(* IEC 61131-3 sources: AXOpen/src/components.mitsubishi.robotics/app/src/IO/PLC_LINE, 7 files *)

(* ---- HwIdentifiers.st ---- *)
TYPE
    HwIdentifiers : WORD
    (
        PROFINET_IO_System_HwID :=	WORD#256,
        TZ535_PN_HwID :=	WORD#260,
        TZ535_PN_In_Out_64_byte_1_In_Out__64_byte_HwID :=	WORD#263,
        TZ535_PN_Rack_HwID :=	WORD#261,
        TZ535_PN_TZ535_PN_HwID :=	WORD#262,
        TZ535_PN_TZ535_PN_2D_TZ535_PNPROFINET_IO_HwID :=	WORD#264,
        TZ535_PN_TZ535_PN_profinet_HwID :=	WORD#257,
        TZ535_PN_TZ535_PN_profinet_Port_1_HwID :=	WORD#258,
        TZ535_PN_TZ535_PN_profinet_Port_2_HwID :=	WORD#259,
        plc_line_HwID :=	WORD#32,
        plc_line_Rail_0_HwID :=	WORD#265,
        plc_line_plc_line_HwID :=	WORD#48,
        plc_line_plc_line__plc_line_HwID :=	WORD#49,
        plc_line_plc_line_CPU_display_1_HwID :=	WORD#54,
        plc_line_plc_line_CPU_exec_unit_1_HwID :=	WORD#52,
        plc_line_plc_line_Card_reader_writer_1_HwID :=	WORD#51,
        plc_line_plc_line_DP_interface_1_HwID :=	WORD#60,
        plc_line_plc_line_LicenseManager_1_HwID :=	WORD#42,
        plc_line_plc_line_OPC_UA_1_HwID :=	WORD#117,
        plc_line_plc_line_PROFINET_interface_2_HwID :=	WORD#72,
        plc_line_plc_line_PROFINET_interface_2_Port_1_HwID :=	WORD#73,
        plc_line_plc_line_Virtual_communication_interface_HwID :=	WORD#135,
        plc_line_plc_line_plc_line_HwID :=	WORD#50,
        plc_line_plc_line_profinet_x1_HwID :=	WORD#64,
        plc_line_plc_line_profinet_x1_Port1_HwID :=	WORD#65,
        plc_line_plc_line_profinet_x1_Port2_HwID :=	WORD#66,

        NONE := WORD#0
    );
END_TYPE

(* ---- HwInputs.st ---- *)
TYPE
	HwInputs : STRUCT
		TZ535_PN_In_Out_64_byte_1 AT %B0 : ARRAY[0..63] OF BYTE;
	END_STRUCT;
END_TYPE

(* ---- HwOutputs.st ---- *)
TYPE
	HwOutputs : STRUCT
		TZ535_PN_In_Out_64_byte_1 AT %B0 : ARRAY[0..63] OF BYTE;
	END_STRUCT;
END_TYPE

(* ---- PlcInputs.st ---- *)
TYPE
	PlcInputs : STRUCT
		TZ535_PN_In_Out_64_byte_1 : ARRAY[0..63] OF BYTE;
	END_STRUCT;
END_TYPE

(* ---- PlcOutputs.st ---- *)
TYPE
	PlcOutputs : STRUCT
		TZ535_PN_In_Out_64_byte_1 : ARRAY[0..63] OF BYTE;
	END_STRUCT;
END_TYPE

(* ---- CopyInputs.st ---- *)
FUNCTION CopyInputs
	VAR_EXTERNAL
		HwInputs : HwInputs;
		PlcInputs : PlcInputs;
	END_VAR
	PlcInputs.TZ535_PN_In_Out_64_byte_1[0] := HwInputs.TZ535_PN_In_Out_64_byte_1[0];
	PlcInputs.TZ535_PN_In_Out_64_byte_1[1] := HwInputs.TZ535_PN_In_Out_64_byte_1[1];
	PlcInputs.TZ535_PN_In_Out_64_byte_1[2] := HwInputs.TZ535_PN_In_Out_64_byte_1[2];
	PlcInputs.TZ535_PN_In_Out_64_byte_1[3] := HwInputs.TZ535_PN_In_Out_64_byte_1[3];
	PlcInputs.TZ535_PN_In_Out_64_byte_1[4] := HwInputs.TZ535_PN_In_Out_64_byte_1[4];
	PlcInputs.TZ535_PN_In_Out_64_byte_1[5] := HwInputs.TZ535_PN_In_Out_64_byte_1[5];
	PlcInputs.TZ535_PN_In_Out_64_byte_1[6] := HwInputs.TZ535_PN_In_Out_64_byte_1[6];
	PlcInputs.TZ535_PN_In_Out_64_byte_1[7] := HwInputs.TZ535_PN_In_Out_64_byte_1[7];
	PlcInputs.TZ535_PN_In_Out_64_byte_1[8] := HwInputs.TZ535_PN_In_Out_64_byte_1[8];
	PlcInputs.TZ535_PN_In_Out_64_byte_1[9] := HwInputs.TZ535_PN_In_Out_64_byte_1[9];
	PlcInputs.TZ535_PN_In_Out_64_byte_1[10] := HwInputs.TZ535_PN_In_Out_64_byte_1[10];
	PlcInputs.TZ535_PN_In_Out_64_byte_1[11] := HwInputs.TZ535_PN_In_Out_64_byte_1[11];
	PlcInputs.TZ535_PN_In_Out_64_byte_1[12] := HwInputs.TZ535_PN_In_Out_64_byte_1[12];
	PlcInputs.TZ535_PN_In_Out_64_byte_1[13] := HwInputs.TZ535_PN_In_Out_64_byte_1[13];
	PlcInputs.TZ535_PN_In_Out_64_byte_1[14] := HwInputs.TZ535_PN_In_Out_64_byte_1[14];
	PlcInputs.TZ535_PN_In_Out_64_byte_1[15] := HwInputs.TZ535_PN_In_Out_64_byte_1[15];
	PlcInputs.TZ535_PN_In_Out_64_byte_1[16] := HwInputs.TZ535_PN_In_Out_64_byte_1[16];
	PlcInputs.TZ535_PN_In_Out_64_byte_1[17] := HwInputs.TZ535_PN_In_Out_64_byte_1[17];
	PlcInputs.TZ535_PN_In_Out_64_byte_1[18] := HwInputs.TZ535_PN_In_Out_64_byte_1[18];
	PlcInputs.TZ535_PN_In_Out_64_byte_1[19] := HwInputs.TZ535_PN_In_Out_64_byte_1[19];
	PlcInputs.TZ535_PN_In_Out_64_byte_1[20] := HwInputs.TZ535_PN_In_Out_64_byte_1[20];
	PlcInputs.TZ535_PN_In_Out_64_byte_1[21] := HwInputs.TZ535_PN_In_Out_64_byte_1[21];
	PlcInputs.TZ535_PN_In_Out_64_byte_1[22] := HwInputs.TZ535_PN_In_Out_64_byte_1[22];
	PlcInputs.TZ535_PN_In_Out_64_byte_1[23] := HwInputs.TZ535_PN_In_Out_64_byte_1[23];
	PlcInputs.TZ535_PN_In_Out_64_byte_1[24] := HwInputs.TZ535_PN_In_Out_64_byte_1[24];
	PlcInputs.TZ535_PN_In_Out_64_byte_1[25] := HwInputs.TZ535_PN_In_Out_64_byte_1[25];
	PlcInputs.TZ535_PN_In_Out_64_byte_1[26] := HwInputs.TZ535_PN_In_Out_64_byte_1[26];
	PlcInputs.TZ535_PN_In_Out_64_byte_1[27] := HwInputs.TZ535_PN_In_Out_64_byte_1[27];
	PlcInputs.TZ535_PN_In_Out_64_byte_1[28] := HwInputs.TZ535_PN_In_Out_64_byte_1[28];
	PlcInputs.TZ535_PN_In_Out_64_byte_1[29] := HwInputs.TZ535_PN_In_Out_64_byte_1[29];
	PlcInputs.TZ535_PN_In_Out_64_byte_1[30] := HwInputs.TZ535_PN_In_Out_64_byte_1[30];
	PlcInputs.TZ535_PN_In_Out_64_byte_1[31] := HwInputs.TZ535_PN_In_Out_64_byte_1[31];
	PlcInputs.TZ535_PN_In_Out_64_byte_1[32] := HwInputs.TZ535_PN_In_Out_64_byte_1[32];
	PlcInputs.TZ535_PN_In_Out_64_byte_1[33] := HwInputs.TZ535_PN_In_Out_64_byte_1[33];
	PlcInputs.TZ535_PN_In_Out_64_byte_1[34] := HwInputs.TZ535_PN_In_Out_64_byte_1[34];
	PlcInputs.TZ535_PN_In_Out_64_byte_1[35] := HwInputs.TZ535_PN_In_Out_64_byte_1[35];
	PlcInputs.TZ535_PN_In_Out_64_byte_1[36] := HwInputs.TZ535_PN_In_Out_64_byte_1[36];
	PlcInputs.TZ535_PN_In_Out_64_byte_1[37] := HwInputs.TZ535_PN_In_Out_64_byte_1[37];
	PlcInputs.TZ535_PN_In_Out_64_byte_1[38] := HwInputs.TZ535_PN_In_Out_64_byte_1[38];
	PlcInputs.TZ535_PN_In_Out_64_byte_1[39] := HwInputs.TZ535_PN_In_Out_64_byte_1[39];
	PlcInputs.TZ535_PN_In_Out_64_byte_1[40] := HwInputs.TZ535_PN_In_Out_64_byte_1[40];
	PlcInputs.TZ535_PN_In_Out_64_byte_1[41] := HwInputs.TZ535_PN_In_Out_64_byte_1[41];
	PlcInputs.TZ535_PN_In_Out_64_byte_1[42] := HwInputs.TZ535_PN_In_Out_64_byte_1[42];
	PlcInputs.TZ535_PN_In_Out_64_byte_1[43] := HwInputs.TZ535_PN_In_Out_64_byte_1[43];
	PlcInputs.TZ535_PN_In_Out_64_byte_1[44] := HwInputs.TZ535_PN_In_Out_64_byte_1[44];
	PlcInputs.TZ535_PN_In_Out_64_byte_1[45] := HwInputs.TZ535_PN_In_Out_64_byte_1[45];
	PlcInputs.TZ535_PN_In_Out_64_byte_1[46] := HwInputs.TZ535_PN_In_Out_64_byte_1[46];
	PlcInputs.TZ535_PN_In_Out_64_byte_1[47] := HwInputs.TZ535_PN_In_Out_64_byte_1[47];
	PlcInputs.TZ535_PN_In_Out_64_byte_1[48] := HwInputs.TZ535_PN_In_Out_64_byte_1[48];
	PlcInputs.TZ535_PN_In_Out_64_byte_1[49] := HwInputs.TZ535_PN_In_Out_64_byte_1[49];
	PlcInputs.TZ535_PN_In_Out_64_byte_1[50] := HwInputs.TZ535_PN_In_Out_64_byte_1[50];
	PlcInputs.TZ535_PN_In_Out_64_byte_1[51] := HwInputs.TZ535_PN_In_Out_64_byte_1[51];
	PlcInputs.TZ535_PN_In_Out_64_byte_1[52] := HwInputs.TZ535_PN_In_Out_64_byte_1[52];
	PlcInputs.TZ535_PN_In_Out_64_byte_1[53] := HwInputs.TZ535_PN_In_Out_64_byte_1[53];
	PlcInputs.TZ535_PN_In_Out_64_byte_1[54] := HwInputs.TZ535_PN_In_Out_64_byte_1[54];
	PlcInputs.TZ535_PN_In_Out_64_byte_1[55] := HwInputs.TZ535_PN_In_Out_64_byte_1[55];
	PlcInputs.TZ535_PN_In_Out_64_byte_1[56] := HwInputs.TZ535_PN_In_Out_64_byte_1[56];
	PlcInputs.TZ535_PN_In_Out_64_byte_1[57] := HwInputs.TZ535_PN_In_Out_64_byte_1[57];
	PlcInputs.TZ535_PN_In_Out_64_byte_1[58] := HwInputs.TZ535_PN_In_Out_64_byte_1[58];
	PlcInputs.TZ535_PN_In_Out_64_byte_1[59] := HwInputs.TZ535_PN_In_Out_64_byte_1[59];
	PlcInputs.TZ535_PN_In_Out_64_byte_1[60] := HwInputs.TZ535_PN_In_Out_64_byte_1[60];
	PlcInputs.TZ535_PN_In_Out_64_byte_1[61] := HwInputs.TZ535_PN_In_Out_64_byte_1[61];
	PlcInputs.TZ535_PN_In_Out_64_byte_1[62] := HwInputs.TZ535_PN_In_Out_64_byte_1[62];
	PlcInputs.TZ535_PN_In_Out_64_byte_1[63] := HwInputs.TZ535_PN_In_Out_64_byte_1[63];
END_FUNCTION

(* ---- CopyOutputs.st ---- *)
FUNCTION CopyOutputs
	VAR_EXTERNAL
		HwOutputs : HwOutputs;
		PlcOutputs : PlcOutputs;
	END_VAR
	HwOutputs.TZ535_PN_In_Out_64_byte_1[0] := PlcOutputs.TZ535_PN_In_Out_64_byte_1[0];
	HwOutputs.TZ535_PN_In_Out_64_byte_1[1] := PlcOutputs.TZ535_PN_In_Out_64_byte_1[1];
	HwOutputs.TZ535_PN_In_Out_64_byte_1[2] := PlcOutputs.TZ535_PN_In_Out_64_byte_1[2];
	HwOutputs.TZ535_PN_In_Out_64_byte_1[3] := PlcOutputs.TZ535_PN_In_Out_64_byte_1[3];
	HwOutputs.TZ535_PN_In_Out_64_byte_1[4] := PlcOutputs.TZ535_PN_In_Out_64_byte_1[4];
	HwOutputs.TZ535_PN_In_Out_64_byte_1[5] := PlcOutputs.TZ535_PN_In_Out_64_byte_1[5];
	HwOutputs.TZ535_PN_In_Out_64_byte_1[6] := PlcOutputs.TZ535_PN_In_Out_64_byte_1[6];
	HwOutputs.TZ535_PN_In_Out_64_byte_1[7] := PlcOutputs.TZ535_PN_In_Out_64_byte_1[7];
	HwOutputs.TZ535_PN_In_Out_64_byte_1[8] := PlcOutputs.TZ535_PN_In_Out_64_byte_1[8];
	HwOutputs.TZ535_PN_In_Out_64_byte_1[9] := PlcOutputs.TZ535_PN_In_Out_64_byte_1[9];
	HwOutputs.TZ535_PN_In_Out_64_byte_1[10] := PlcOutputs.TZ535_PN_In_Out_64_byte_1[10];
	HwOutputs.TZ535_PN_In_Out_64_byte_1[11] := PlcOutputs.TZ535_PN_In_Out_64_byte_1[11];
	HwOutputs.TZ535_PN_In_Out_64_byte_1[12] := PlcOutputs.TZ535_PN_In_Out_64_byte_1[12];
	HwOutputs.TZ535_PN_In_Out_64_byte_1[13] := PlcOutputs.TZ535_PN_In_Out_64_byte_1[13];
	HwOutputs.TZ535_PN_In_Out_64_byte_1[14] := PlcOutputs.TZ535_PN_In_Out_64_byte_1[14];
	HwOutputs.TZ535_PN_In_Out_64_byte_1[15] := PlcOutputs.TZ535_PN_In_Out_64_byte_1[15];
	HwOutputs.TZ535_PN_In_Out_64_byte_1[16] := PlcOutputs.TZ535_PN_In_Out_64_byte_1[16];
	HwOutputs.TZ535_PN_In_Out_64_byte_1[17] := PlcOutputs.TZ535_PN_In_Out_64_byte_1[17];
	HwOutputs.TZ535_PN_In_Out_64_byte_1[18] := PlcOutputs.TZ535_PN_In_Out_64_byte_1[18];
	HwOutputs.TZ535_PN_In_Out_64_byte_1[19] := PlcOutputs.TZ535_PN_In_Out_64_byte_1[19];
	HwOutputs.TZ535_PN_In_Out_64_byte_1[20] := PlcOutputs.TZ535_PN_In_Out_64_byte_1[20];
	HwOutputs.TZ535_PN_In_Out_64_byte_1[21] := PlcOutputs.TZ535_PN_In_Out_64_byte_1[21];
	HwOutputs.TZ535_PN_In_Out_64_byte_1[22] := PlcOutputs.TZ535_PN_In_Out_64_byte_1[22];
	HwOutputs.TZ535_PN_In_Out_64_byte_1[23] := PlcOutputs.TZ535_PN_In_Out_64_byte_1[23];
	HwOutputs.TZ535_PN_In_Out_64_byte_1[24] := PlcOutputs.TZ535_PN_In_Out_64_byte_1[24];
	HwOutputs.TZ535_PN_In_Out_64_byte_1[25] := PlcOutputs.TZ535_PN_In_Out_64_byte_1[25];
	HwOutputs.TZ535_PN_In_Out_64_byte_1[26] := PlcOutputs.TZ535_PN_In_Out_64_byte_1[26];
	HwOutputs.TZ535_PN_In_Out_64_byte_1[27] := PlcOutputs.TZ535_PN_In_Out_64_byte_1[27];
	HwOutputs.TZ535_PN_In_Out_64_byte_1[28] := PlcOutputs.TZ535_PN_In_Out_64_byte_1[28];
	HwOutputs.TZ535_PN_In_Out_64_byte_1[29] := PlcOutputs.TZ535_PN_In_Out_64_byte_1[29];
	HwOutputs.TZ535_PN_In_Out_64_byte_1[30] := PlcOutputs.TZ535_PN_In_Out_64_byte_1[30];
	HwOutputs.TZ535_PN_In_Out_64_byte_1[31] := PlcOutputs.TZ535_PN_In_Out_64_byte_1[31];
	HwOutputs.TZ535_PN_In_Out_64_byte_1[32] := PlcOutputs.TZ535_PN_In_Out_64_byte_1[32];
	HwOutputs.TZ535_PN_In_Out_64_byte_1[33] := PlcOutputs.TZ535_PN_In_Out_64_byte_1[33];
	HwOutputs.TZ535_PN_In_Out_64_byte_1[34] := PlcOutputs.TZ535_PN_In_Out_64_byte_1[34];
	HwOutputs.TZ535_PN_In_Out_64_byte_1[35] := PlcOutputs.TZ535_PN_In_Out_64_byte_1[35];
	HwOutputs.TZ535_PN_In_Out_64_byte_1[36] := PlcOutputs.TZ535_PN_In_Out_64_byte_1[36];
	HwOutputs.TZ535_PN_In_Out_64_byte_1[37] := PlcOutputs.TZ535_PN_In_Out_64_byte_1[37];
	HwOutputs.TZ535_PN_In_Out_64_byte_1[38] := PlcOutputs.TZ535_PN_In_Out_64_byte_1[38];
	HwOutputs.TZ535_PN_In_Out_64_byte_1[39] := PlcOutputs.TZ535_PN_In_Out_64_byte_1[39];
	HwOutputs.TZ535_PN_In_Out_64_byte_1[40] := PlcOutputs.TZ535_PN_In_Out_64_byte_1[40];
	HwOutputs.TZ535_PN_In_Out_64_byte_1[41] := PlcOutputs.TZ535_PN_In_Out_64_byte_1[41];
	HwOutputs.TZ535_PN_In_Out_64_byte_1[42] := PlcOutputs.TZ535_PN_In_Out_64_byte_1[42];
	HwOutputs.TZ535_PN_In_Out_64_byte_1[43] := PlcOutputs.TZ535_PN_In_Out_64_byte_1[43];
	HwOutputs.TZ535_PN_In_Out_64_byte_1[44] := PlcOutputs.TZ535_PN_In_Out_64_byte_1[44];
	HwOutputs.TZ535_PN_In_Out_64_byte_1[45] := PlcOutputs.TZ535_PN_In_Out_64_byte_1[45];
	HwOutputs.TZ535_PN_In_Out_64_byte_1[46] := PlcOutputs.TZ535_PN_In_Out_64_byte_1[46];
	HwOutputs.TZ535_PN_In_Out_64_byte_1[47] := PlcOutputs.TZ535_PN_In_Out_64_byte_1[47];
	HwOutputs.TZ535_PN_In_Out_64_byte_1[48] := PlcOutputs.TZ535_PN_In_Out_64_byte_1[48];
	HwOutputs.TZ535_PN_In_Out_64_byte_1[49] := PlcOutputs.TZ535_PN_In_Out_64_byte_1[49];
	HwOutputs.TZ535_PN_In_Out_64_byte_1[50] := PlcOutputs.TZ535_PN_In_Out_64_byte_1[50];
	HwOutputs.TZ535_PN_In_Out_64_byte_1[51] := PlcOutputs.TZ535_PN_In_Out_64_byte_1[51];
	HwOutputs.TZ535_PN_In_Out_64_byte_1[52] := PlcOutputs.TZ535_PN_In_Out_64_byte_1[52];
	HwOutputs.TZ535_PN_In_Out_64_byte_1[53] := PlcOutputs.TZ535_PN_In_Out_64_byte_1[53];
	HwOutputs.TZ535_PN_In_Out_64_byte_1[54] := PlcOutputs.TZ535_PN_In_Out_64_byte_1[54];
	HwOutputs.TZ535_PN_In_Out_64_byte_1[55] := PlcOutputs.TZ535_PN_In_Out_64_byte_1[55];
	HwOutputs.TZ535_PN_In_Out_64_byte_1[56] := PlcOutputs.TZ535_PN_In_Out_64_byte_1[56];
	HwOutputs.TZ535_PN_In_Out_64_byte_1[57] := PlcOutputs.TZ535_PN_In_Out_64_byte_1[57];
	HwOutputs.TZ535_PN_In_Out_64_byte_1[58] := PlcOutputs.TZ535_PN_In_Out_64_byte_1[58];
	HwOutputs.TZ535_PN_In_Out_64_byte_1[59] := PlcOutputs.TZ535_PN_In_Out_64_byte_1[59];
	HwOutputs.TZ535_PN_In_Out_64_byte_1[60] := PlcOutputs.TZ535_PN_In_Out_64_byte_1[60];
	HwOutputs.TZ535_PN_In_Out_64_byte_1[61] := PlcOutputs.TZ535_PN_In_Out_64_byte_1[61];
	HwOutputs.TZ535_PN_In_Out_64_byte_1[62] := PlcOutputs.TZ535_PN_In_Out_64_byte_1[62];
	HwOutputs.TZ535_PN_In_Out_64_byte_1[63] := PlcOutputs.TZ535_PN_In_Out_64_byte_1[63];
END_FUNCTION
